TYPE DB_r134a :
STRUCT
	id: DINT;
	timestamp: DT;
	Temperatur: STRING(45);
	Enthalpie: STRING(45);
	Druck: STRING(45);
END_STRUCT
END_TYPE

(* stored: Version 1.1.0.1, ProductVersion 3.1.4018.5
   DUT DB_r134a: Id {104427af-734f-4a2b-b8ae-006d16d5d762} *)
